FUNCTION_BLOCK FB_HeaterControl (* Basic Function Block Type *)
  (* Standard: 61499-2 *)
  (* Version 0.0, 2014-5-4, wildai, nxtControl GmbH, Template *)
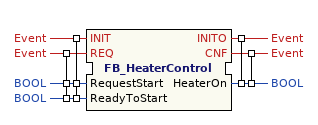
  EVENT_INPUT
    INIT WITH RequestStart, ReadyToStart; (* Initialization Request *)
    REQ WITH RequestStart, ReadyToStart; (* Normal Execution Request *)
  END_EVENT
  EVENT_OUTPUT
    INITO WITH HeaterOn; (* Initialization Confirm *)
    CNF WITH HeaterOn; (* Execution Confirmation *)
  END_EVENT
  VAR_INPUT
    RequestStart : BOOL;
    ReadyToStart : BOOL;
  END_VAR
  VAR_OUTPUT
    HeaterOn : BOOL; (* Output event qualifier *)
  END_VAR
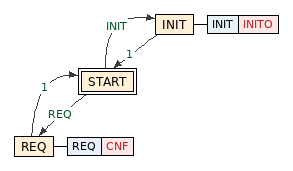
  EC_STATES
    START; (* Initial State *)
    INIT : INIT -> INITO; (* Initialization *)
    REQ : REQ -> CNF; (* Normal execution *)
  END_STATES
  EC_TRANSITIONS
    START TO INIT := INIT;
    INIT TO START := 1;
    START TO REQ := REQ;
    REQ TO START := 1;
  END_TRANSITIONS
  ALGORITHM INIT IN ST: (* Initialization algorithm *)
;

HeaterOn := FALSE;
  END_ALGORITHM
  ALGORITHM REQ IN ST: (* Normally executed algorithm *)
;

IF RequestStart AND ReadyToStart THEN
	HeaterOn := TRUE;
ELSE
	HeaterOn := FALSE;
END_IF;
  END_ALGORITHM
END_FUNCTION_BLOCK
